// TIA Portal V18 export
TYPE "SubProcessParameterP020_ShW"
// stored: IsFailsafeCompliant false
   STRUCT
      Reserved : Bool;
   END_STRUCT;
END_TYPE
